PROGRAM Stn053_27_EmptyPuckStorageMainMergePrestopRed
VAR
	{attribute 'TcLinkToOSO' := '.iPuckPresent   :=  <0,1,3>TIIB[N46S00 (AL1332)]^N46S05 (AL2341)^TxPDO^input byte 0;
		.iBufferFull   :=  <0,1,3>TIIB[N46S00 (AL1332)]^N46S05 (AL2341)^TxPDO^input byte 2;
		.oStopLower :=  <0,1,1>TIIB[N46S00 (AL1332)]^N46S02 (EX260)^RxPDO^output byte 1'}
	fbConvStop: FB_ConvStop;
END_VAR

//  This code instantiates a component that is implimented as a common function block
//    Note that I/O is linked directly to I/O variables inside the named instance

gStn053_27_EmptyPuckStorageMainMergePrestopRed.ConvRunning  := gConsumed_SafetyInterfaceConv.MtrRunning.Enc056Mtr06;

fbConvStop(
	pStn := ADR(gStn053),
	pCmp := ADR(gStn053_27_EmptyPuckStorageMainMergePrestopRed),
	pUpstreamStop := 0,
	pStateTraceBuffer := ADR(gStn053_StateTraceBuffer),
	pStateTraceFifo := ADR(gStn053_StateTraceFifo),
	pStats := ADR(gStn053_02_Stats));

END_PROGRAM

(* stored: Version 1.1.0.1, ProductVersion 3.1.4024.6
   POU Stn053_27_EmptyPuckStorageMainMergePrestopRed: Id {74491f48-908f-46a5-8064-f81210e29171}, SpecialFunc None *)
